ABB RobotStudio station: Vision_HG_20240221-183452.rsstn

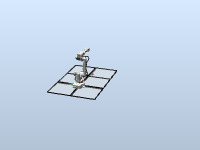
Station Station (saved by RobotStudio 6.8.8148.134)
Controller 2600-507493New
  mechanical unit ROB_1: IRB2600_20_165__02, 6 joints, base frame (0, 0, 0) mm
Layout (positions relative to the parent item):
  - IRB2600_20_165__02 [mechanism, from Robots\IRB2600_20_165_G_02.rslib] at (0, 0, 0) mm; joint values [0, 0, 0, 0, 0.5236, 0] (rad or m)
  - 框架_2 [frame] at (695.76, -308.93, 242.8) mm, rotated rx -4.43 ry -84.98 rz 46.15 deg
